FUNCTION_BLOCK TEventHandler
IMPLEMENTS
    IEventHandler_OnExecutionAborted,
    IEventHandler_OnExecutionFailed
VAR_INPUT
END_VAR
VAR_OUTPUT
END_VAR
VAR
    _AbortedEventRaised : BOOL;
    _FailedEventRaised : BOOL;
    _EventMessage : T_MaxString;
END_VAR

PROPERTY AbortedEventRaised : BOOL
GET
AbortedEventRaised := _AbortedEventRaised;
END_GET
SET
_AbortedEventRaised := AbortedEventRaised;
END_SET
END_PROPERTY

PROPERTY EventMessage : T_MaxString
GET
END_GET
SET
END_SET
END_PROPERTY

PROPERTY FailedEventRaised : BOOL
GET
FailedEventRaised := _FailedEventRaised;
END_GET
SET
_FailedEventRaised := FailedEventRaised;
END_SET
END_PROPERTY

METHOD OnExecutionAborted
VAR_INPUT
	Message	: Tc2_System.T_MaxString;
END_VAR
_AbortedEventRaised := TRUE;
_EventMessage := Message;
END_METHOD

METHOD OnExecutionFailed
VAR_INPUT
	Message	: Tc2_System.T_MaxString;
END_VAR
_FailedEventRaised := TRUE;
_EventMessage := Message;
END_METHOD

END_FUNCTION_BLOCK

(* stored: Version 1.1.0.1, ProductVersion 3.1.4024.3
   POU TEventHandler: Id {446b80c4-412f-43c3-b3df-49796ca9b150}, SpecialFunc None
   Property AbortedEventRaised: Id {380c722c-ddf8-434d-acb4-13d6bb013408}
   Get Get: Id {153a1b11-7655-42a9-9cca-e68fb826407b}
   Set Set: Id {15dac4d4-4ed2-4530-8493-86572b19ed4c}
   Property EventMessage: Id {1623a7a6-d174-4447-a320-a4160363ceea}
   Get Get: Id {206d8337-4b37-4d70-81a2-bc512455b389}
   Set Set: Id {b09b8163-efaa-4fd1-a418-7b23b8fe5678}
   Property FailedEventRaised: Id {baf314f0-2868-46c2-bf52-35702b2bd54d}
   Get Get: Id {9a9eb52b-fb7c-4514-8a3f-1adc36a2f8b6}
   Set Set: Id {feec5263-e5ea-47fe-ad67-f996d40f4d56}
   Method OnExecutionAborted: Id {43f4685c-b454-47b8-b453-3776181a57de}
   Method OnExecutionFailed: Id {7b6e5be1-7bfd-4bcc-a964-b69bd7943de1} *)
